{attribute 'qualified_only'}
{attribute 'strict'}
TYPE eTransitionType :
(
    None := 0,
    Linear := 1,
    Exponential := 2,
    S_Type := 3
);
END_TYPE

(* stored: Version 1.1.0.1
   DUT eTransitionType: Id {a1c6b4db-4aa1-095c-02b5-b8aef9374a51} *)
